// This function has been automatically generated from the project information.
{attribute 'signature_flag' := '1073741824'}
{attribute 'TcGenerated'}
{attribute 'no-analysis'}
FUNCTION F_GetCompany : WSTRING
VAR_INPUT
	
END_VAR

F_GetCompany := "www.peterzerlauth.com";

END_FUNCTION

(* stored: Version 1.1.0.1
   POU F_GetCompany: Id {4e58c019-b49c-455f-b3c9-476a56eaf3cf}, SpecialFunc None *)
